PROGRAM MAIN
VAR
	nCounter : DINT ;
END_VAR

END_PROGRAM

(* stored: Version 1.1.0.1, ProductVersion 3.1.4024.13
   POU MAIN: Id {5bfb7f6e-1311-403e-b2ed-88510c09bdb8}, SpecialFunc None *)
